PROGRAM c05_CustomFBs
VAR_INPUT
	Enable 			: BOOL;
END_VAR
VAR_OUTPUT
	isInited : BOOL;
END_VAR
VAR
	sACN_Com : FB_sACN_UDP_Communicator; //Transit variable representing the UDP communicator for sACN.

	sACN_Sender_U111: FB_sACN_Source_SBSPM;//Custom Functionality FB
	
	sACN_Receiver_U555:	FB_sACN_ReceiverAndMerger_SBSPM;
	
	LastReceivedPacketNum : UINT;
	i : UINT;
END_VAR

sACN_Com(NetworkAdapterNum:= E_NetworkAdapters.SLOT_N02, //<- Change if it is necessary
			 ReconnectTime:= T#5M, 
			 BindedToNetworkAdapter=> , 
			 BindedAdapterInfo=> );
			 
IF NOT isInited THEN
	isInited := TRUE;
	
	sACN_Receiver_U555.BindExternalDmxArray(Term06.DmxLightFixture_Left);
END_IF

sACN_Sender_U111(
	sAcnCommunicator:= sACN_Com, 
	Enable:= Enable, 
	SourceName:= 'BeckhoffPLC ControlPanel U111', 
	CID:= Tc2_Utilities.STRING_TO_GUID('3566cea5-b4a4-48fc-aa02-cd84a65f0a88'),  //Generated by https://www.guidgenerator.com/
	sAcnUniverse:= 111, 
	PacketPriority:= 100, 
	SendingPeriod:= T#100MS, 
	SentPackets=> );

sACN_Receiver_U555(
	sAcnCommunicator:= sACN_Com, 
	Enable:= Enable,
	sAcnUniverse:= 555,
	MergeRule:= );

END_PROGRAM

(* stored: Version 1.1.0.1
   POU c05_CustomFBs: Id {428b9a48-28ed-4692-8610-f71c3498164b}, SpecialFunc None *)
